IF bPersistentCheckpointStart THEN
	bPersistentCheckpointInFlight := TRUE;
	nPersistentCheckpointStartedGeneration :=
		nPersistentCheckpointRequestGeneration;
	fCheckpointPositionX := GVL_Persistent.fLastPositionX;
	fCheckpointPositionY := GVL_Persistent.fLastPositionY;
	bCheckpointValidX := GVL_Persistent.bLastPositionValidX;
	bCheckpointValidY := GVL_Persistent.bLastPositionValidY;
ELSIF bPersistentCheckpointInFlight AND
	NOT fbWritePersistentData.BUSY THEN
	bPersistentCheckpointInFlight := FALSE;
	nPersistentCheckpointCompletedGeneration :=
		nPersistentCheckpointStartedGeneration;
	bPersistentCheckpointPending :=
		nPersistentCheckpointCompletedGeneration <>
		nPersistentCheckpointRequestGeneration;
	IF fbWritePersistentData.ERR THEN
		bPersistentPositionSaved := FALSE;
		bPersistentPositionSaveError := TRUE;
		nPersistentPositionSaveErrorID :=
			fbWritePersistentData.ERRID;
	ELSE
		bPersistentPositionSaved := TRUE;
		bPersistentPositionSaveError := FALSE;
		nPersistentPositionSaveErrorID := 0;
		nPersistentPositionCheckpointCounter :=
			nPersistentPositionCheckpointCounter + 1;
	END_IF
END_IF

bPersistentPositionSaveBusy :=
	bPersistentCheckpointPending OR
	bPersistentCheckpointInFlight OR
	fbWritePersistentData.BUSY;

// Home and reset are one-shot commands
stMoveCommandX.bHome := FALSE;
stMoveCommandY.bHome := FALSE;
stMoveCommandX.bReset := FALSE;
stMoveCommandY.bReset := FALSE;
stMoveCommandX.bSavePosition := FALSE;
stMoveCommandY.bSavePosition := FALSE;
stMoveCommandX.bRestorePosition := FALSE;
stMoveCommandY.bRestorePosition := FALSE;

END_PROGRAM
